% RSLogix 500 project Automated Nut Sorting & Packaging System (PLC Controls).RSS, saved by version 8.30.00.16 %
PROJECT "P2"    % processor: Bul.1763 MicroLogix 1100 Series B %

PROGRAM FILES
  LAD 2   4 rungs
  LAD 3 "IO"  8 rungs
  LAD 4 "CTRL"  6 rungs
  LAD 5 "CYCLE"  5 rungs

DATA FILES
  O0 OUTPUT  4 elements
  I1 INPUT  6 elements
  S2 STATUS  66 elements
  B3 BINARY  1 elements
  T4 TIMER  1 elements
  C5 COUNTER  1 elements
  R6 CONTROL  1 elements
  N7 INTEGER  1 elements
  F8 FLOAT  1 elements

LADDER 2
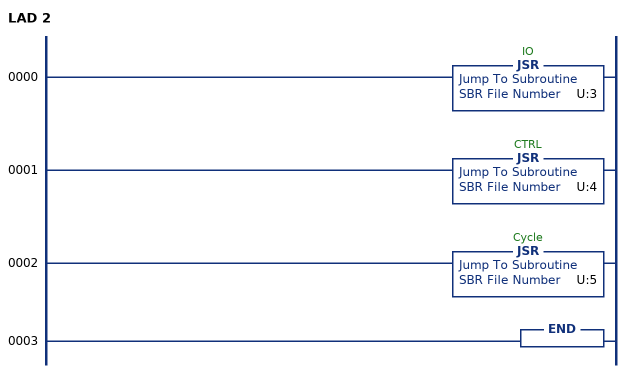
% Rung: 0 %
SOR JSR U:3 EOR
%   U:3  "IO" %
% Rung: 1 %
SOR JSR U:4 EOR
%   U:4  "CTRL" %
% Rung: 2 %
SOR JSR U:5 EOR
%   U:5  "Cycle" %
% Rung: 3 %
SOR END EOR

LADDER 3 "IO"
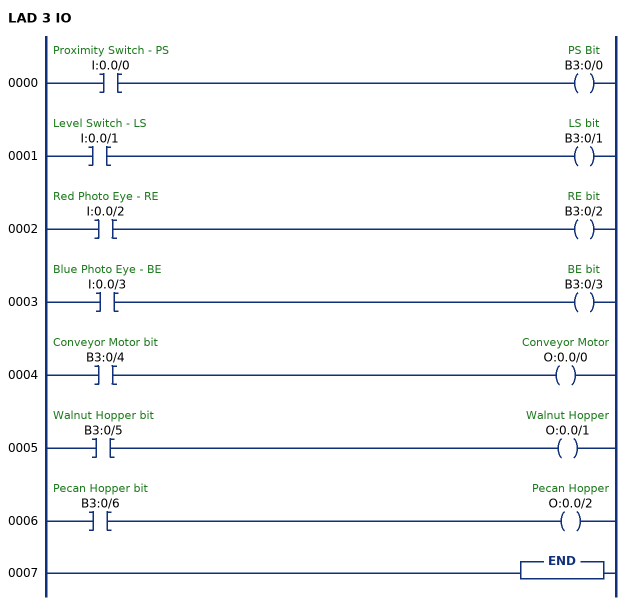
% Rung: 0 %
SOR XIC I:0.0/0 OTE B3:0/0 EOR
%   I:0.0/0  "Proximity Switch - PS" %
%   B3:0/0  "PS Bit" %
% Rung: 1 %
SOR XIC I:0.0/1 OTE B3:0/1 EOR
%   I:0.0/1  "Level Switch - LS" %
%   B3:0/1  "LS bit" %
% Rung: 2 %
SOR XIC I:0.0/2 OTE B3:0/2 EOR
%   I:0.0/2  "Red Photo Eye - RE" %
%   B3:0/2  "RE bit" %
% Rung: 3 %
SOR XIC I:0.0/3 OTE B3:0/3 EOR
%   I:0.0/3  "Blue Photo Eye - BE" %
%   B3:0/3  "BE bit" %
% Rung: 4 %
SOR XIC B3:0/4 OTE O:0.0/0 EOR
%   B3:0/4  "Conveyor Motor bit" %
%   O:0.0/0  "Conveyor Motor" %
% Rung: 5 %
SOR XIC B3:0/5 OTE O:0.0/1 EOR
%   B3:0/5  "Walnut Hopper bit" %
%   O:0.0/1  "Walnut Hopper" %
% Rung: 6 %
SOR XIC B3:0/6 OTE O:0.0/2 EOR
%   B3:0/6  "Pecan Hopper bit" %
%   O:0.0/2  "Pecan Hopper" %
% Rung: 7 %
SOR END EOR

LADDER 4 "CTRL"
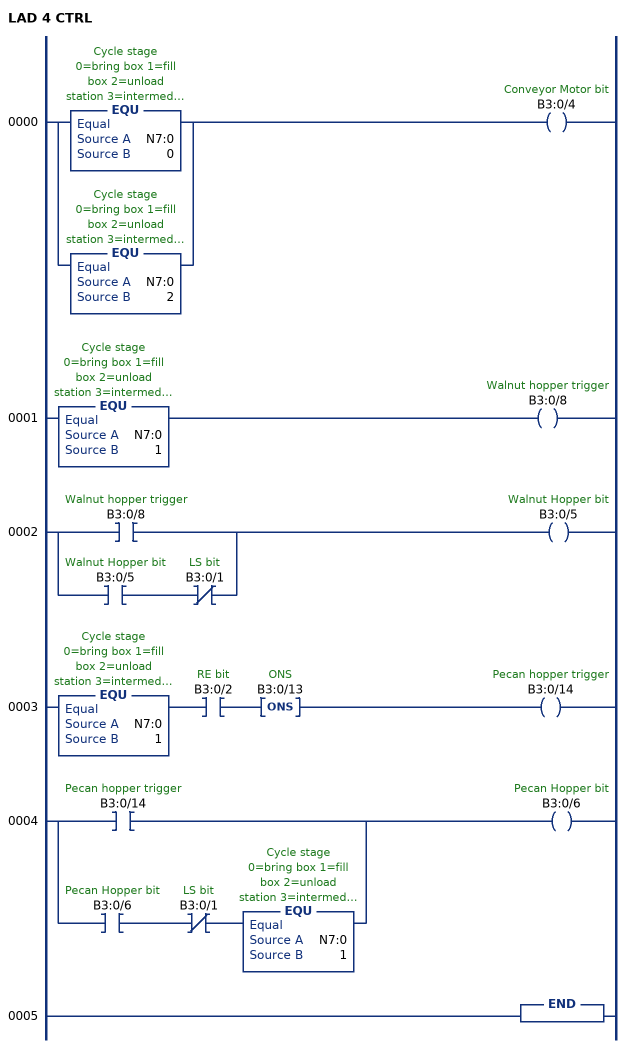
% Rung: 0 %
SOR BST EQU N7:0 0 NXB EQU N7:0 2 BND OTE B3:0/4 EOR
%   N7:0  "Cycle stage 0=bring box 1=fill box 2=unload station 3=intermediate" %
%   B3:0/4  "Conveyor Motor bit" %
% Rung: 1 %
SOR EQU N7:0 1 OTE B3:0/8 EOR
%   N7:0  "Cycle stage 0=bring box 1=fill box 2=unload station 3=intermediate" %
%   B3:0/8  "Walnut hopper trigger" %
% Rung: 2 %
SOR BST XIC B3:0/8 NXB XIC B3:0/5 XIO B3:0/1 BND OTE B3:0/5 EOR
%   B3:0/8  "Walnut hopper trigger" %
%   B3:0/5  "Walnut Hopper bit" %
%   B3:0/1  "LS bit" %
% Rung: 3 %
SOR EQU N7:0 1 XIC B3:0/2 ONS B3:0/13 OTE B3:0/14 EOR
%   N7:0  "Cycle stage 0=bring box 1=fill box 2=unload station 3=intermediate" %
%   B3:0/2  "RE bit" %
%   B3:0/13  "ONS" %
%   B3:0/14  "Pecan hopper trigger" %
% Rung: 4 %
SOR BST XIC B3:0/14 NXB XIC B3:0/6 XIO B3:0/1 EQU N7:0 1 BND OTE B3:0/6 EOR
%   B3:0/14  "Pecan hopper trigger" %
%   B3:0/6  "Pecan Hopper bit" %
%   B3:0/1  "LS bit" %
%   N7:0  "Cycle stage 0=bring box 1=fill box 2=unload station 3=intermediate" %
% Rung: 5 %
SOR END EOR

LADDER 5 "CYCLE"
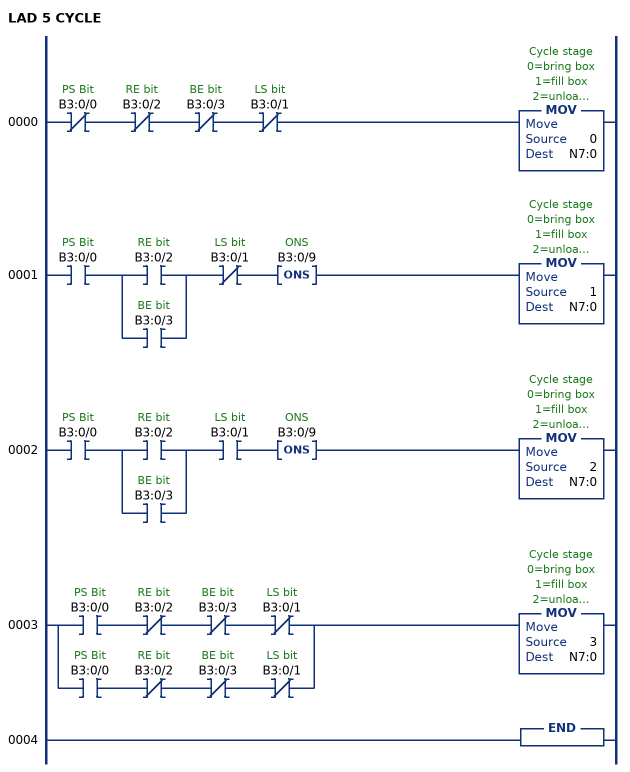
% Rung: 0 %
SOR XIO B3:0/0 XIO B3:0/2 XIO B3:0/3 XIO B3:0/1 MOV 0 N7:0 EOR
%   B3:0/0  "PS Bit" %
%   B3:0/2  "RE bit" %
%   B3:0/3  "BE bit" %
%   B3:0/1  "LS bit" %
%   N7:0  "Cycle stage 0=bring box 1=fill box 2=unload station 3=intermediate" %
% Rung: 1 %
SOR XIC B3:0/0 BST XIC B3:0/2 NXB XIC B3:0/3 BND XIO B3:0/1 ONS B3:0/9 MOV 1 N7:0 EOR
%   B3:0/0  "PS Bit" %
%   B3:0/2  "RE bit" %
%   B3:0/3  "BE bit" %
%   B3:0/1  "LS bit" %
%   B3:0/9  "ONS" %
%   N7:0  "Cycle stage 0=bring box 1=fill box 2=unload station 3=intermediate" %
% Rung: 2 %
SOR XIC B3:0/0 BST XIC B3:0/2 NXB XIC B3:0/3 BND XIC B3:0/1 ONS B3:0/9 MOV 2 N7:0 EOR
%   B3:0/0  "PS Bit" %
%   B3:0/2  "RE bit" %
%   B3:0/3  "BE bit" %
%   B3:0/1  "LS bit" %
%   B3:0/9  "ONS" %
%   N7:0  "Cycle stage 0=bring box 1=fill box 2=unload station 3=intermediate" %
% Rung: 3 %
SOR BST XIC B3:0/0 XIO B3:0/2 XIO B3:0/3 XIO B3:0/1 NXB XIC B3:0/0 XIO B3:0/2 XIO B3:0/3 XIO B3:0/1 BND MOV 3 N7:0 EOR
%   B3:0/0  "PS Bit" %
%   B3:0/2  "RE bit" %
%   B3:0/3  "BE bit" %
%   B3:0/1  "LS bit" %
%   N7:0  "Cycle stage 0=bring box 1=fill box 2=unload station 3=intermediate" %
% Rung: 4 %
SOR END EOR

OTHER DOCUMENTED ADDRESSES
  B3:0/7  "ONS"
  T4:0  "Coveyor Start delay"
  T4:1  "Pecan hopper delay"
